// TIA Portal V17 export
FUNCTION "数学运算指令" : Void   // FC, LAD
{ S7_Optimized_Access := 'TRUE' }
VERSION : 0.1
// stored: AutoNumber true, IsIECCheckEnabled false, SetENOAutomatically false
BEGIN

REGION Network 1
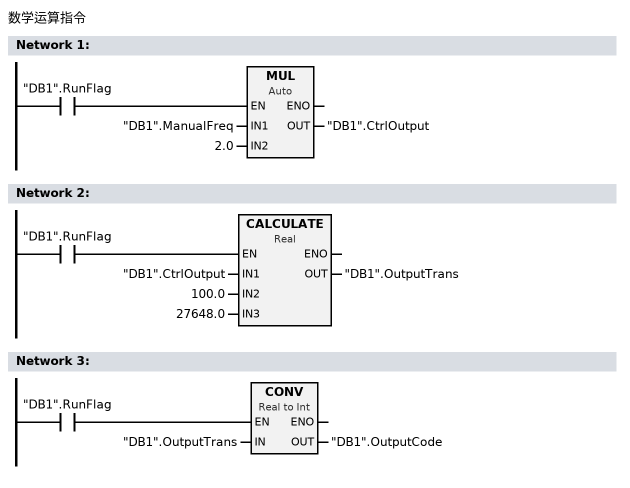
   RUNG wire#powerrail
      Contact( "DB1".RunFlag )
      { S7_GenerateENO := "TRUE" } Mul(in1 := "DB1".ManualFreq, in2 := 2.0, out => "DB1".CtrlOutput)
   END_RUNG
   // the same network as SCL:
   IF "DB1".RunFlag THEN "DB1".CtrlOutput := "DB1".ManualFreq * 2.0; END_IF;
END_REGION

REGION Network 2
   RUNG wire#powerrail
      Contact( "DB1".RunFlag )
      { S7_Templates := "SrcType := Real"; S7_GenerateENO := "TRUE"; S7_Expression := "(IN1/IN2)*IN3" } Calculate(in1 := "DB1".CtrlOutput, in2 := 100.0, in3 := 27648.0, out => "DB1".OutputTrans)
   END_RUNG
   // the same network as SCL:
   IF "DB1".RunFlag THEN "DB1".OutputTrans := ("DB1".CtrlOutput/100.0)*27648.0; END_IF;
END_REGION

REGION Network 3
   RUNG wire#powerrail
      Contact( "DB1".RunFlag )
      { S7_Templates := "[SrcType := Real, DestType := Int]"; S7_GenerateENO := "TRUE" } Convert(in := "DB1".OutputTrans, out => "DB1".OutputCode)
   END_RUNG
   // the same network as SCL:
   IF "DB1".RunFlag THEN "DB1".OutputCode := REAL_TO_INT("DB1".OutputTrans); END_IF;
END_REGION
END_FUNCTION
